      # second byte is '7'?
      if (list_of_bytes[2] != 55):
          return False
      end

      return True
  end

  def is_FLT_autorelease_in_progress(list_of_bytes):

      # list length is not 2
      if (list_of_bytes[0] != 2):
          return False
      end

      # first byte is '1'?
      if (list_of_bytes[1] != 49):
          return False
      end

      # second byte is '1'?
      if (list_of_bytes[2] != 49):
          return False
      end

      return True

  end

  def is_FLT_overcurrent(list_of_bytes):

      # list length is not 2
      if (list_of_bytes[0] != 2):
          return False
      end

      # first byte is '1'?
      if (list_of_bytes[1] != 49):
          return False
      end

      # second byte is '4'?
      if (list_of_bytes[2] != 52):
          return False
      end

      return True

  end

  def is_FLT_autorelease_completed(list_of_bytes):

      # list length is not 2
      if (list_of_bytes[0] != 2):
          return False
      end

      # first byte is '1'?
      if (list_of_bytes[1] != 49):
          return False
      end

      # second byte is '5'?
      if (list_of_bytes[2] != 53):
          return False
      end

      return True

  end

  def rq_set_var(var_name, var_value, gripper_socket="1"):

      var_name_string = ""

      if (var_name == ACT):
          var_name_string = "ACT"
      elif (var_name == GTO):
          var_name_string = "GTO"
      elif (var_name == ATR):
          var_name_string = "ATR"
      elif (var_name == ARD):
          var_name_string = "ARD"
      elif (var_name == FOR):
          var_name_string = "FOR"
      elif (var_name == SPE):
          var_name_string = "SPE"
      elif (var_name == POS):
          var_name_string = "POS"
      elif (var_name == LBP):
          var_name_string = "LBP"
      elif (var_name == LRD):
          var_name_string = "LRD"
      elif (var_name == LBL):
          var_name_string = "LBL"
      elif (var_name == LGN):
          var_name_string = "LGN"
      elif (var_name == MSC):
          var_name_string = "MSC"
      elif (var_name == MOD):
          var_name_string = "MOD"
      end

      rq_acquire_gripper_socket(gripper_socket)
      socket_set_var(var_name_string, var_value, gripper_socket)
      sync()
      ack = socket_read_byte_list(3, gripper_socket)
      rq_release_gripper_socket(gripper_socket)

      sync()

      while(is_not_ack(ack)):
          rq_acquire_gripper_socket(gripper_socket)
          socket_set_var(var_name_string , var_value, gripper_socket)
          sync()
          ack = socket_read_byte_list(3, gripper_socket)
          rq_release_gripper_socket(gripper_socket)

          sync()
      end
  end


  def rq_get_var(var_name, nbr_bytes, gripper_socket="1"):
      rq_acquire_gripper_socket(gripper_socket)

      if (var_name == FLT):
          socket_send_string("GET FLT", gripper_socket)
      elif (var_name == OBJ):
          socket_send_string("GET OBJ", gripper_socket)
      elif (var_name == STA):
          socket_send_string("GET STA", gripper_socket)
      elif (var_name == PRE):
          socket_send_string("GET PRE", gripper_socket)
      elif (var_name == GTO):
          socket_send_string("GET GTO", gripper_socket)
      else:
      end

      sync()

      var_value = socket_read_byte_list(nbr_bytes, gripper_socket)

      rq_release_gripper_socket(gripper_socket)

      sync()

      return var_value
  end

  def rq_is_object_validated(gripper_selected, gripper_socket="1"):
      if(gripper_selected):
          if(rq_is_object_detected(gripper_socket)):
              return True
          else:
              return False
          end
      else:
          return True
      end
  end

  ############################################
  # normalized functions (maps 0-100 to 0-255)
  ############################################
  def rq_set_force_norm(force_norm, gripper_socket="1"):
      force_gripper = norm_to_gripper(force_norm)
      rq_set_force(force_gripper, gripper_socket)
  end

  def rq_set_speed_norm(speed_norm, gripper_socket="1"):
      speed_gripper = norm_to_gripper(speed_norm)
      rq_set_speed(speed_gripper, gripper_socket)
  end

  def rq_move_norm(pos_norm, gripper_socket="1"):
      pos_gripper = norm_to_gripper(pos_norm)
      rq_move(pos_gripper, gripper_socket)
  end

  def rq_move_and_wait_norm(pos_norm, gripper_socket="1"):
      pos_gripper = norm_to_gripper(pos_norm)
      rq_move_and_wait(pos_gripper, gripper_socket)
  end

  def rq_set_pos_norm(pos_norm, gripper_socket="1"):
      pos_gripper = norm_to_gripper(pos_norm)
      rq_set_pos(pos_gripper, gripper_socket)
  end

  def rq_current_pos_norm(gripper_socket="1"):
      pos_gripper = rq_current_pos(gripper_socket)
      pos_norm = gripper_to_norm(pos_gripper)
      return pos_norm
  end

  def gripper_to_norm(value_gripper):
      value_norm = (value_gripper / 255) * 100
      return floor(value_norm)
  end

  def norm_to_gripper(value_norm):
      value_gripper = (value_norm / 100) * 255
      return ceil(value_gripper)
  end

  def rq_get_position():
      return rq_current_pos_norm()
  end

  def rq_gripper_led_on(gripper_socket="1"):
      rq_set_var(LBP,0, gripper_socket)
  end

  def rq_gripper_led_off(gripper_socket="1"):
      rq_set_var(LBP,1, gripper_socket)
      rq_set_var(LRD,0, gripper_socket)
      rq_set_var(LBL,0, gripper_socket)
      rq_set_var(LGN,0, gripper_socket)
  end

  def rq_gripper_led_force_red(gripper_socket="1"):
      rq_set_var(LBP,1, gripper_socket)
      rq_set_var(LRD,1, gripper_socket)
      rq_set_var(LBL,0, gripper_socket)
      rq_set_var(LGN,0, gripper_socket)
  end

  def rq_gripper_led_force_blue(gripper_socket="1"):
      rq_set_var(LBP,1, gripper_socket)
      rq_set_var(LRD,0, gripper_socket)
      rq_set_var(LBL,1, gripper_socket)
      rq_set_var(LGN,0, gripper_socket)
  end

  def rq_gripper_led_force_green(gripper_socket="1"):
      rq_set_var(LBP,1, gripper_socket)
      rq_set_var(LRD,0, gripper_socket)
      rq_set_var(LBL,0, gripper_socket)
      rq_set_var(LGN,1, gripper_socket)
  end

  def rq_gripper_led_force_purple(gripper_socket="1"):
      rq_set_var(LBP,1, gripper_socket)
      rq_set_var(LRD,1, gripper_socket)
      rq_set_var(LBL,1, gripper_socket)
      rq_set_var(LGN,0, gripper_socket)
  end

  ############################################
  # mm/inches functions
  ############################################
  gripper_closed_norm = [100, 100, 100, 100]
  gripper_open_norm = [0, 0, 0, 0]
  gripper_closed_mm = [0, 0, 0, 0]
  gripper_open_mm = [50, 50, 50, 50]

  def rq_current_pos_mm(gripper_socket=1):
      pos_gripper = rq_current_pos(gripper_socket)
      pos_mm = gripper_to_mm(pos_gripper, gripper_socket)
      return round_value_2_dec(pos_mm)
  end

  def rq_current_pos_inches(gripper_socket=1):
      pos_gripper = rq_current_pos(gripper_socket)
      pos_mm = gripper_to_mm(pos_gripper, gripper_socket)
      pos_in = pos_mm / 25.4
      return round_value_2_dec(pos_in)
  end

  def rq_move_mm(pos_mm, gripper_socket=1):
      pos_gripper = mm_to_gripper(pos_mm, gripper_socket)
      rq_move(pos_gripper, gripper_socket)
  end

  def rq_move_and_wait_mm(pos_mm, gripper_socket=1):
      pos_gripper = mm_to_gripper(pos_mm, gripper_socket)
      rq_move_and_wait(pos_gripper, gripper_socket)
  end

  def rq_move_inches(pos_in, gripper_socket=1):
      pos_mm = pos_in * 25.4
      rq_move_mm(pos_mm, gripper_socket)
  end

  def rq_move_and_wait_inches(pos_in, gripper_socket=1):
      pos_mm = pos_in * 25.4
      rq_move_and_wait_mm(pos_mm, gripper_socket)
  end

  def get_closed_norm(gripper_socket):
      return gripper_closed_norm[gripper_socket - 1]
  end

  def get_open_norm(gripper_socket):
      return gripper_open_norm[gripper_socket - 1]
  end

  def get_closed_mm(gripper_socket):
      return gripper_closed_mm[gripper_socket - 1]
  end

  def get_open_mm(gripper_socket):
      return gripper_open_mm[gripper_socket - 1]
  end

  def set_closed_norm(closed_norm, gripper_socket):
      gripper_closed_norm[gripper_socket - 1] = closed_norm
  end

  def set_open_norm(open_norm, gripper_socket):
      gripper_open_norm[gripper_socket - 1] = open_norm
  end

  def set_closed_mm(closed_mm, gripper_socket):
      gripper_closed_mm[gripper_socket - 1] = closed_mm
  end

  def set_open_mm(open_mm, gripper_socket):
      gripper_open_mm[gripper_socket - 1] = open_mm
  end

  def gripper_to_mm(value_gripper, gripper_socket):
      closed_norm = get_closed_norm(gripper_socket)
      open_norm = get_open_norm(gripper_socket)
      closed_mm = get_closed_mm(gripper_socket)
      open_mm = get_open_mm(gripper_socket)

      value_norm = (value_gripper / 255) * 100

      slope = (closed_mm - open_mm) / (closed_norm - open_norm)
      value_mm = slope * (value_norm - closed_norm) + closed_mm

      if (value_mm > open_mm):
          value_mm_limited = open_mm
      elif (value_mm < closed_mm):
          value_mm_limited = closed_mm
      else:
          value_mm_limited = value_mm
      end

      return value_mm_limited
  end

  def mm_to_gripper(value_mm, gripper_socket):
      closed_norm = get_closed_norm(gripper_socket)
      open_norm = get_open_norm(gripper_socket)
      closed_mm = get_closed_mm(gripper_socket)
      open_mm = get_open_mm(gripper_socket)

      slope = (closed_norm - open_norm) / (closed_mm - open_mm)
      value_norm = (value_mm - closed_mm) * slope + closed_norm

      value_gripper = value_norm * 255 / 100

      if (value_gripper > 255):
          value_gripper_limited = 255
      elif (value_gripper < 0):
          value_gripper_limited = 0
      else:
          value_gripper_limited = round_value(value_gripper)
      end

      return value_gripper_limited
  end

  def round_value(value):
      value_mod = value % 1

      if(value_mod < 0.5):
          return floor(value)
      else:
          return ceil(value)
      end
  end

  def round_value_2_dec(value):
      value_x_100 = value * 100
      value_x_100_rounded = round_value(value_x_100)
      return value_x_100_rounded / 100
  end

  def clear_socket_buffer(gripper_socket="1", read_timeout = 0.1):
    byte_in_buffer = socket_read_byte_list(1, gripper_socket, read_timeout)

    while(byte_in_buffer[0] >= 1):
        byte_in_buffer = socket_read_byte_list(1, gripper_socket, read_timeout)
    end
  end

  def rq_set_gripper_socket_acquire_option(enabled=False):
      gripper_socket_acquire_option = enabled

      if(not enabled):
          gripper_1_socket_acquired = False
          gripper_2_socket_acquired = False
          gripper_3_socket_acquired = False
          gripper_4_socket_acquired = False
      end
  end

  def rq_acquire_gripper_socket(gripper_socket="1"):
      if(gripper_socket_acquire_option):
          rq_wait_gripper_socket_released(gripper_socket)
          enter_critical
              rq_set_gripper_socket_acquired(gripper_socket, True)
          exit_critical

          clear_socket_buffer(gripper_socket, 0.002)

          sync()
      end
  end

  def rq_release_gripper_socket(gripper_socket="1"):
      if(gripper_socket_acquire_option):
          rq_set_gripper_socket_acquired(gripper_socket, False)

          sync()
      end
  end

  def rq_set_gripper_socket_acquired(gripper_socket="1", acquired=False):
      if(gripper_socket == "1"):
          gripper_1_socket_acquired = acquired
      elif(gripper_socket == "2"):
          gripper_2_socket_acquired = acquired
      elif(gripper_socket == "3"):
          gripper_3_socket_acquired = acquired
      elif(gripper_socket == "4"):
          gripper_4_socket_acquired = acquired
      end
  end

  def rq_get_gripper_socket_acquired(gripper_socket="1"):
      if(gripper_socket == "1"):
          return gripper_1_socket_acquired
      elif(gripper_socket == "2"):
          return gripper_2_socket_acquired
      elif(gripper_socket == "3"):
          return gripper_3_socket_acquired
      elif(gripper_socket == "4"):
          return gripper_4_socket_acquired
      end

      sync()
  end

  def rq_wait_gripper_socket_released(gripper_socket="1"):
      while(rq_get_gripper_socket_acquired(gripper_socket)):
          sync()
      end

      sync()
  end

  def rq_gripper_id_to_ascii(gripper_id):
      if(gripper_id == "1"):
          return 57
      elif(gripper_id == "2"):
          return 50
      elif(gripper_id == "3"):
          return 51
      elif(gripper_id == "4"):
          return 52
      end
  end

  def scale(value, rawRange, scaledRange):
      def computeSlope(inputRange, outputRange):
          outputRangeDelta = outputRange[1] - outputRange[0]
          inputRangeDelta = inputRange[1] - inputRange[0]

          if (inputRangeDelta == 0):
              return 0
          else:
              return outputRangeDelta / inputRangeDelta
          end
      end

      def computeIntercept(slope, inputRange, outputRange):
          return outputRange[0] - (slope * inputRange[0])
      end

      def clipScaledValue(outputScaledValue, outputRange):
          if (outputRange[0] < outputRange[1]):
              return clipWhenLowerLimitIsLessThanHigher(outputScaledValue, outputRange)
          else:
              return clipWhenLowerLimitIsGreaterThanHigherLimit(outputScaledValue, outputRange)
          end
      end

      def clipWhenLowerLimitIsGreaterThanHigherLimit(outputScaledValue, outputRange):
          if (outputScaledValue < outputRange[1]):
              return outputRange[1]
          elif (outputScaledValue > outputRange[0]):
              return outputRange[0]
          else:
              return outputScaledValue
          end
      end

      def clipWhenLowerLimitIsLessThanHigher(outputScaledValue, outputRange):
          if (outputScaledValue < outputRange[0]):
              return outputRange[0]
          elif (outputScaledValue > outputRange[1]):
              return outputRange[1]
          else:
              return outputScaledValue
          end
      end

      slope = computeSlope(rawRange, scaledRange)
      intercept = computeIntercept(slope, rawRange, scaledRange)
      scaledValue = slope * value + intercept
      return clipScaledValue(scaledValue, scaledRange)
  end

  def limit(value, range):
      return scale(value, range, range)
  end


  rq_obj_detect = 0
  rq_init_comm_if_connected(9, "1")
  rq_init_comm_if_connected(2, "2")
  rq_init_comm_if_connected(3, "3")
  rq_init_comm_if_connected(4, "4")
  rq_print_connected_grippers()
  connectivity_checked = [-1,-1,-1,-1]
  status_checked = [-1,-1,-1,-1]
  current_speed = [-1,-1,-1,-1]
  current_force = [-1,-1,-1,-1]
  set_closed_norm(100.0, 1)
  set_open_norm(0.0, 1)
  set_closed_mm(0.0, 1)
  set_open_mm(50.0, 1)
  set_closed_norm(100.0, 2)
  set_open_norm(0.0, 2)
  set_closed_mm(0.0, 2)
  set_open_mm(50.0, 2)
  set_closed_norm(100.0, 3)
  set_open_norm(0.0, 3)
  set_closed_mm(0.0, 3)
  set_open_mm(50.0, 3)
  set_closed_norm(100.0, 4)
  set_open_norm(0.0, 4)
  set_closed_mm(0.0, 4)
  set_open_mm(50.0, 4)
  rq_current_limit_enabled = False
  # end: URCap Installation Node
  # begin: URCap Installation Node
  #   Source: PART LOCALIZATION WITH SICK PLOC2D, 2.3.0, SICK AG - Developed by Nimalendiran Kailasanathan
  #   Type: PLOC2D HELP
  global PLOC2D_CONNECTION = "NOT CONNECTED"
  global ANYFEEDER_CONNECTION = "NOT CONNECTED"
  global PLOC2D_STATUS = "Job(s) not located."
  global PLOC_LOCATED = False
  global PLOC_IS_WITHIN_REACH = False
  global PLOC2D_JOB_ID = 0
  global PLOC2D_LOCATE_TRIALS = 0
  global PLOC2D_URPose = p[0,0,0,0,0,0]
   def ploc2d_wrist(pose,jRefPose,activeTCP):
			jJoints=get_inverse_kin(pose,jRefPose,1e-10,1e-10,activeTCP)
			return jJoints
	end
   def ploc_wrist_pose(pose,jRefPose,activeTCP):
			jJoints=get_inverse_kin(pose,jRefPose,1e-10,1e-10,activeTCP)
			finalPose=get_forward_kin(jJoints,activeTCP)
			return finalPose
	end
		def PLOC2D_SendString(PLOC2D_string): #Function to send a string over the socket. INPUT: string to send
			PLOC2D_sent=False
			#textmsg("string",PLOC2D_string)
			PLOC2D_sent=socket_send_string(PLOC2D_string, "Sick_Ploc_Socket")
			sleep(0.01)
			if not PLOC2D_sent:
	  			popup("Failed to send string message","Message Transmission Failure",False,True,blocking=True)
			end
		end
		def PLOC2D_SendStringToAnyfeeder(PLOC2D_AnyfeederString): #Function to send a string over the socket. INPUT: string to send
			PLOC2D_AnyfeederSent=False
			#textmsg("string",PLOC2D_AnyfeederString)
			PLOC2D_AnyfeederSent=socket_send_string(PLOC2D_AnyfeederString, "Anyfeeder_Socket")
			sleep(0.01)
			if not PLOC2D_AnyfeederSent:
	  			popup("Failed to send string message","Message Transmission Failure",False,True,blocking=True)
			end
		end
		def PLOC2D_convertPose(PoseFromPLOC): #Function to convert the frames from a list with millimiters, and RPY angles in degrees data (as returned by PLOC2D_) to a pose variable (meters, radians, axis angle notation) as used by the UR robot. INPUT=list (length 6) with frame format from PLOC2D_ (mm, RPY angles in degrees). OUTPUT=UR robot pose.
			PLOC2D_rotRPY=[0,0,0]
			PLOC2D_rotRPY[0]=d2r(PoseFromPLOC[5])  #Rx
			PLOC2D_rotRPY[1]=d2r(PoseFromPLOC[6])  #Ry
			PLOC2D_rotRPY[2]=d2r(PoseFromPLOC[7])  #Rz
			PLOC2D_rotVec=rpy2rotvec(PLOC2D_rotRPY)
			PLOC2D_convertedPose=p[PoseFromPLOC[2]/1000,PoseFromPLOC[3]/1000,PoseFromPLOC[4]/1000,PLOC2D_rotVec[0],PLOC2D_rotVec[1],PLOC2D_rotVec[2]]
			return PLOC2D_convertedPose
		end
		def PLOC2D_LocatePart(PLOC2D_command): #Function to ask PLOC2D_ to locate a part. INPUT= string PLOC2D_ job Alias. OUTPUT=list with received part result data
			#PLOC2D_command = "Run.Locate,1"
           PLOC2D_located = "Run.Locate.Ok"
			#textmsg("sent",PLOC2D_command)
			PLOC2D_SendString(PLOC2D_command)
       	#sleep(0.2)
			PLOC2D_receivedPartMsg=socket_read_string("Sick_Ploc_Socket","","",False,120)
					#textmsg(PLOC2D_receivedPartMsg)
			PLOC2D_delimiter = ","
			PLOC2D_l=0
			l_token =0
			PLOC2D_ok=-1
			PLOC2D_data=[0,0,0,0,0,0,0,0,0]
			PLOC2D_pos=0
			PLOC2D_token=" "
			s_length = str_len(PLOC2D_receivedPartMsg)
			first=True
			while PLOC2D_ok!= 0:
				PLOC2D_pos = str_find(PLOC2D_receivedPartMsg,PLOC2D_delimiter)
				if PLOC2D_pos==-1:
					PLOC2D_token = PLOC2D_receivedPartMsg
					PLOC2D_ok=0
					#textmsg(PLOC2D_data)
				else:
					PLOC2D_token = str_sub(PLOC2D_receivedPartMsg,0,PLOC2D_pos)
					l_token = str_len(PLOC2D_token)
					PLOC2D_receivedPartMsg=str_sub(PLOC2D_receivedPartMsg,l_token+1,s_length)
				end
				if first:
					first=False
					if PLOC2D_token == PLOC2D_located:
						PLOC2D_data[0]=1
					else:
						PLOC2D_data[0]=0
						break
					end
				end
				if PLOC2D_l == 1:
					PLOC2D_data[1] = to_num(PLOC2D_token)
				elif PLOC2D_l == 4:
					PLOC2D_data[2] = to_num(PLOC2D_token)
				elif PLOC2D_l == 5:
					PLOC2D_data[3] = to_num(PLOC2D_token)
				elif PLOC2D_l == 6:
					PLOC2D_data[4] = to_num(PLOC2D_token)
				elif PLOC2D_l == 7:
					PLOC2D_data[5] = to_num(PLOC2D_token)
				elif PLOC2D_l == 8:
					PLOC2D_data[6] = to_num(PLOC2D_token)
				elif PLOC2D_l == 9:
					PLOC2D_data[7] = to_num(PLOC2D_token)
				elif PLOC2D_l == 3:
					PLOC2D_data[8] = to_num(PLOC2D_token)
				end
				PLOC2D_l=PLOC2D_l+1
			end
			return PLOC2D_data
		end
		def PLOC2D_extractPose(PLOC2D_PartData):  #Function extracting a meaningful pose from the part result data obtained from PLOC.
			PLOC2D_correctionFrame=PLOC2D_PartData
			PLOC2D_correctionFrame[2]=PLOC2D_PartData[2]/1
			PLOC2D_correctionFrame[3]=PLOC2D_PartData[3]/1
			PLOC2D_correctionFrame[4]=PLOC2D_PartData[4]/1
			PLOC2D_URPose=PLOC2D_convertPose(PLOC2D_correctionFrame)
			return PLOC2D_URPose
		end
		def PLOC2D_getCorrectedPickPose(PLOC2D_PartData,PLOC_AlignmentF):
			PLOC2D_correctionFrame=PLOC2D_extractPose(PLOC2D_PartData)
			PLOC2D_correctedFrame=pose_trans(PLOC_AlignmentF,PLOC2D_correctionFrame)
			#textmsg(PLOC2D_correctedFrame)
			return PLOC2D_correctedFrame
		end
		def Connect_To_ANYFEEDER(PLOC2D_ip,PLOC2D_port): #Function to establish socket connection with PLOC
			PLOC2D_AnyfeederConnected = False
			PLOC2D_AnyfeederCounter=0
			while not PLOC2D_AnyfeederConnected and (PLOC2D_AnyfeederCounter<100):
	  			PLOC2D_AnyfeederConnected=socket_open(PLOC2D_ip,PLOC2D_port,"Anyfeeder_Socket")
	  			PLOC2D_AnyfeederCounter=PLOC2D_AnyfeederCounter+1
			end
			if PLOC2D_AnyfeederCounter>=100:
	  			popup("Connection to anyfeeder failed","Time out",False,True,blocking=True)
	  			halt
			else:
	  			#textmsg("Connected to Anyfeeder")
				ANYFEEDER_CONNECTION = "Connected to Anyfeeder" 			end
		end
		def Connect_To_PLOC(PLOC2D_ip,PLOC2D_port): #Function to establish socket connection with PLOC
			PLOC2D_Connected = False
			PLOC2D_counter=0
			while not PLOC2D_Connected and (PLOC2D_counter<100):
	  			PLOC2D_Connected=socket_open(PLOC2D_ip,PLOC2D_port,"Sick_Ploc_Socket")
	  			PLOC2D_counter=PLOC2D_counter+1
			end
			if PLOC2D_counter>=100:
	  			popup("Connection to PLOC failed","Time out",False,True,blocking=True)
	  			halt
			else:
	  			#textmsg("Connected to PLOC")
				PLOC2D_CONNECTION = "Connected to PLOC2D_" 			end
		end
		def DISCONNECT_To_PLOC(): #Function to disconnect socket connection with PLOC
			socket_close("Sick_Ploc_Socket")
		end
		def DISCONNECT_To_ANYFEEDER(): #Function to disconnect socket connection with PLOC
			socket_close("Anyfeeder_Socket")
		end
		def PLOC2D_sendToAnyfeed(PLOC2D_AnyfeederCommand): #Function to ask PLOC2D_ to locate a part. INPUT= string PLOC2D_ job Alias. OUTPUT=list with received part result data
			PLOC2D_SendStringToAnyfeeder(PLOC2D_AnyfeederCommand)
       	#sleep(0.2)
			PLOC2D_AnyfeederReceivedPartMsg=socket_read_string("Anyfeeder_Socket","","",False,120)
			#textmsg(PLOC2D_AnyfeederReceivedPartMsg)
			return PLOC2D_AnyfeederReceivedPartMsg
		end
  # end: URCap Installation Node
  $ 1 "BeforeStart"
  $ 2 "open_socket≔socket_open('192.168.65.102',50000,'ur5e_pc')"
  global open_socket=socket_open("192.168.65.102",50000,"ur5e_pc")
  $ 3 "Loop open_socket≟ False "
  while (open_socket ==   False  ):
    $ 4 "open_socket≔socket_open('192.168.65.102',50000,'ur5e_pc')"
    global open_socket=socket_open("192.168.65.102",50000,"ur5e_pc")
  end
  while (True):
    $ 5 "Robot Program"
    $ 8 "If open_socket≟ True "
    if (open_socket ==   True  ):
      $ 9 "string"
      $ 10 "'read string'"
      # 'read string'
      $ 11 "str≔socket_read_string('ur5e_pc')"
      global str=socket_read_string("ur5e_pc")
      $ 12 "Loop str≟''"
      while (str == ""):
        $ 13 "str≔socket_read_string('ur5e_pc')"
        global str=socket_read_string("ur5e_pc")
        $ 14 "Wait: 0.01"
        sleep(0.01)
      end
      $ 15 "'send string'"
      # 'send string'
      $ 16 "was_send≔socket_send_string('ACK','ur5e_pc')"
      global was_send=socket_send_string("ACK","ur5e_pc")
      $ 17 "Loop was_send≟ False "
      while (was_send ==   False  ):
        $ 18 "was_send≔socket_send_string('ACK','ur5e_pc')"
        global was_send=socket_send_string("ACK","ur5e_pc")
        $ 19 "Wait: 0.01"
        sleep(0.01)
      end
      $ 20 "Wait: 0.01"
      sleep(0.01)
      $ 21 "integer"
      $ 22 "'read int'"
      # 'read int'
      $ 23 "data≔socket_read_binary_integer(1,'ur5e_pc')"
      global data=socket_read_binary_integer(1,"ur5e_pc")
      $ 24 "Loop data[0]≟0"
      while (data[0] == 0):
        $ 25 "data≔socket_read_binary_integer(1,'ur5e_pc')"
        global data=socket_read_binary_integer(1,"ur5e_pc")
        $ 26 "Wait: 0.01"
        sleep(0.01)
      end
      $ 27 "'send int'"
      # 'send int'
      $ 28 "was_send≔socket_send_int(9,'ur5e_pc')"
      global was_send=socket_send_int(9,"ur5e_pc")
      $ 29 "Loop was_send≟ False "
      while (was_send ==   False  ):
        $ 30 "was_send≔socket_send_int(9,'ur5e_pc')"
        global was_send=socket_send_int(9,"ur5e_pc")
        $ 31 "Wait: 0.01"
        sleep(0.01)
      end
      $ 32 "Wait: 0.01"
      sleep(0.01)
      $ 33 "integer array"
      $ 34 "'read Int array'"
      # 'read Int array'
      $ 35 "array_size≔3"
      global array_size=3
      $ 36 "data3≔socket_read_binary_integer(array_size,'ur5e_pc')"
      global data3=socket_read_binary_integer(array_size,"ur5e_pc")
      $ 37 "Loop data3[0]≟0"
      while (data3[0] == 0):
        $ 38 "data3≔socket_read_binary_integer(array_size,'ur5e_pc')"
        global data3=socket_read_binary_integer(array_size,"ur5e_pc")
        $ 39 "Wait: 0.01"
        sleep(0.01)
      end
      $ 40 "'send int array'"
      # 'send int array'
      $ 41 "int_array≔[4, 5, 6]"
      global int_array=[4, 5, 6]
      $ 42 "str_int≔to_str(int_array)"
      global str_int=to_str(int_array)
      $ 43 "was_send≔socket_send_string(str_int,'ur5e_pc')"
      global was_send=socket_send_string(str_int,"ur5e_pc")
      $ 44 "Loop was_send≟ False "
      while (was_send ==   False  ):
        $ 45 "was_send≔socket_send_string(str_int,'ur5e_pc')"
        global was_send=socket_send_string(str_int,"ur5e_pc")
        $ 46 "Wait: 0.01"
        sleep(0.01)
      end
      $ 47 "Wait: 0.01"
      sleep(0.01)
      $ 48 "float"
      $ 49 "'get one float'"
      # 'get one float'
      $ 50 "data4≔socket_read_ascii_float(1,'ur5e_pc')"
      global data4=socket_read_ascii_float(1,"ur5e_pc")
      $ 51 "Loop data4[0]≟0"
      while (data4[0] == 0):
        $ 52 "data4≔socket_read_ascii_float(1,'ur5e_pc')"
        global data4=socket_read_ascii_float(1,"ur5e_pc")
        $ 53 "Wait: 0.01"
        sleep(0.01)
      end
      $ 54 "'send array of floats'"
      # 'send array of floats'
      $ 55 "send_floats≔8.8"
      global send_floats=8.8
      $ 56 "str_floats≔to_str(send_floats)"
      global str_floats=to_str(send_floats)
      $ 57 "was_send≔socket_send_string(str_floats,'ur5e_pc')"
      global was_send=socket_send_string(str_floats,"ur5e_pc")
      $ 58 "Loop was_send≟ False "
      while (was_send ==   False  ):
        $ 59 "was_send≔socket_send_string(str_floats,'ur5e_pc')"
        global was_send=socket_send_string(str_floats,"ur5e_pc")
        $ 60 "Wait: 0.01"
        sleep(0.01)
      end
      $ 61 "float array"
      $ 62 "'get array of floats'"
      # 'get array of floats'
      $ 63 "data2≔socket_read_ascii_float(3,'ur5e_pc')"
      global data2=socket_read_ascii_float(3,"ur5e_pc")
      $ 64 "Loop data2[0]≟0"
      while (data2[0] == 0):
        $ 65 "data2≔socket_read_ascii_float(3,'ur5e_pc')"
        global data2=socket_read_ascii_float(3,"ur5e_pc")
        $ 66 "Wait: 0.01"
        sleep(0.01)
      end
      $ 67 "'send array of floats'"
      # 'send array of floats'
      $ 68 "send_floats2≔[4.4, 5.5, 6.6]"
      global send_floats2=[4.4, 5.5, 6.6]
      $ 69 "str_floats≔to_str(send_floats2)"
      global str_floats=to_str(send_floats2)
      $ 70 "was_send≔socket_send_string(str_floats,'ur5e_pc')"
      global was_send=socket_send_string(str_floats,"ur5e_pc")
      $ 71 "Loop was_send≟ False "
      while (was_send ==   False  ):
        $ 72 "was_send≔socket_send_string(str_floats,'ur5e_pc')"
        global was_send=socket_send_string(str_floats,"ur5e_pc")
        $ 73 "Wait: 0.01"
        sleep(0.01)
      end
      $ 74 "socket_close('ur5e_pc')"
      socket_close("ur5e_pc")
      $ 75 "Halt"
      halt
    end
  end
end
